% RSLogix 500 project job 8.RSS, saved by version 10.00.00.00 %
PROJECT "UNTITLED"    % processor: Bul.1763 MicroLogix 1100 Series B %

PROGRAM FILES
  LAD 2   5 rungs

DATA FILES
  O0 OUTPUT  4 elements
  I1 INPUT  6 elements
  S2 STATUS  66 elements
  B3 BINARY  1 elements
  T4 TIMER  1 elements
  C5 COUNTER  1 elements
  R6 CONTROL  1 elements
  N7 INTEGER  1 elements
  F8 FLOAT  1 elements

LADDER 2
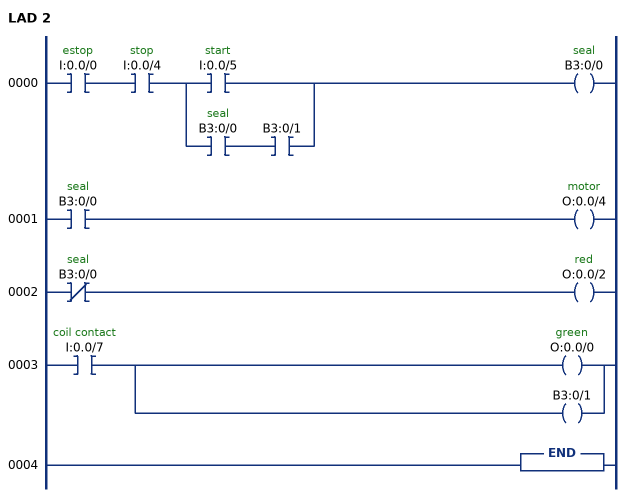
% Rung: 0 %
SOR XIC I:0.0/0 XIC I:0.0/4 BST XIC I:0.0/5 NXB XIC B3:0/0 XIC B3:0/1 BND OTE B3:0/0 EOR
%   I:0.0/0  "estop" %
%   I:0.0/4  "stop" %
%   I:0.0/5  "start" %
%   B3:0/0  "seal" %
% Rung: 1 %
SOR XIC B3:0/0 OTE O:0.0/4 EOR
%   B3:0/0  "seal" %
%   O:0.0/4  "motor" %
% Rung: 2 %
SOR XIO B3:0/0 OTE O:0.0/2 EOR
%   B3:0/0  "seal" %
%   O:0.0/2  "red" %
% Rung: 3 %
SOR XIC I:0.0/7 BST OTE O:0.0/0 NXB OTE B3:0/1 BND EOR
%   I:0.0/7  "coil contact" %
%   O:0.0/0  "green" %
% Rung: 4 %
SOR END EOR

OTHER DOCUMENTED ADDRESSES
  B30:0/0  B
